FUNCTION_BLOCK SlowCounter EXTENDS TcoCore.TcoTask
VAR
    Counter : INT;
    _await : fbAwait;
END_VAR

IF Execute() THEN
    IF _await.Delay(T#250MS) THEN
        Counter := Counter + 1;
    END_IF

    DoneWhen(Counter = 100);
END_IF

(*~
    <docu>
        <summary>
            Restores this instance to the Ready state. Can be called explicitly or from within one of the restore mechanisms.
            <para>
                See also <see cref="PlcDocu.TcoCore.TcoTask.AutoRestorable()"/>
            </para>
        </summary>
    </docu>
~*)
METHOD Restore : ITcoRestorable
SUPER^.Restore();
Counter := 0;
END_METHOD

END_FUNCTION_BLOCK

(* stored: Version 1.1.0.1, ProductVersion 3.1.4024.6
   POU SlowCounter: Id {0fa0c7c4-2a30-0cb7-2afc-736b941f5319}, SpecialFunc None
   Method Restore: Id {407e378a-e722-0999-0be5-fa3a7b67bfd1} *)
